// TIA Portal V16 export
// export: Created 2023-03-29T11:05:04.9469687Z, ExportSetting WithDefaults, DisplayName Totally Integrated Automation Portal, DisplayVersion V16 Update 6, DisplayName TIA Portal Version Control Interface, DisplayVersion V16 Update 2, DisplayName TIA Portal Openness, DisplayVersion V16 Update 6, DisplayName STEP 7 Professional, DisplayVersion V16 Update 6, DisplayName STEP 7 Safety, DisplayVersion V16, DisplayName WinCC Advanced, DisplayVersion V16 Update 6
VAR_GLOBAL   // PLC tag table "Z12"
   isReadyZ12 AT %M86.5 : Bool;
   inputAwariaMomentZ12 AT %M86.1 : Bool;
   inputZamkniętaZ12 AT %M86.3 : Bool;
   imputRuchZ12 AT %M86.4 : Bool;
   setSVMO_Z12 AT %M86.6 : Bool;   // Znacznik polecenia otwórz w trybie automat
   inputmodeAutZ12 AT %M86.7 : Bool;   // Znacznik trybu pracy 1=Aut, 0=Rem
   inputAumalokalneZ12 AT %M87.6 : Bool;
   inputAumaautomatZ12 AT %M87.7 : Bool;
   inputAumagotowośćZ12 AT %M88.0 : Bool;
   inputAumaawariaZ12 AT %M88.1 : Bool;
   setSVMC_Z12 AT %M88.2 : Bool;   // Znacznik polecenia zamknij w trybie automat
   CMD_Open_Z12 AT %M33.5 : Bool;   // załącz otwieranie Z11
   CMD_Close_Z12 AT %M33.6 : Bool;   // załącz zamykanie Z11
   CMD_Awaria_Z12 AT %M91.1 : Bool;   // Awaria zbiorcza
   setAlarm_Moment_Z12 AT %M91.4 : Bool;   // znacznik alarmu od momentówki w trybie zdalnym (aut/mamnual)
   bitH_Alarm_Z12 AT %M97.0 : Bool;   // Alarm - kopia sygału z instancji DB10
   bitH_Open_Z12 AT %M97.1 : Bool;   // Otwarta - kopia sygału z instancji DB10
   bitH_REM_Z12 AT %M97.2 : Bool;   // Zdalne - kopia sygału z instancji DB10
   bitH_Close_Z12 AT %M97.3 : Bool;   // Zamknięta - kopia sygału z instancji DB10
   bitH_Opening_Z12 AT %M97.4 : Bool;   // sygnał otwórz- kopia sygału z instancji DB10
   bitH_Closing_Z12 AT %M97.5 : Bool;   // sygnał zamknij- kopia sygału z instancji DB10
   bitH_Res_Z12 AT %M97.6 : Bool;   // sygnał reset - kopia sygału z instancji DB10
   bitH_Aut_Man_Z12 AT %M97.7 : Bool;   // sygnał aut=1, manual =0 - kopia sygału z instancji DB10
   inputOtwartaZ12 AT %M86.2 : Bool;
   Byte_Status_Z12 AT %MB97 : Byte;   // status napędu
END_VAR
